FUNCTION_BLOCK Equipo_Motor_No_Rev

VAR_INPUT
PE 	  					  : BOOL; (*Parada deemergencia*)
Lock_Out 				  : BOOL;
Conf_Marcha 			  : BOOL; (*Confirmacion de Marcha *)
Modo_Automatico           : BOOL;
Cmd_Auto         		  : BOOL;
Habilitado  			  : BOOL;
T_Discrepancia            : TIME;
END_VAR

VAR_OUTPUT
	Marcha_Equipo	 	  : BOOL;
	Marcha_Ok  				  : BOOL;
	Estado					  : INT;
	Alr_Discrepancia		  : BOOL;	
	Alr_LockOut        		  : BOOL;
END_VAR

VAR_IN_OUT
	Cmd_Man 				  : BOOL;
	Alarma				      : BOOL;
	Horas_Parciales			  : DINT;
	Horas_Totales		 	  : DINT;
	Reset_Horas         	  : BOOL;
	Reset_Alarma		      : BOOL;
END_VAR

VAR_TEMP
	Reset_Cmd_Auto 		      : BOOL;
	Aux_Limpieza		      : TIME;
END_VAR

VAR_STAT
	Cmd_Auto_Directa		  : BOOL;
	FP_Reset				  : R_TRIG;
	FN_Parada_Auto			  : F_TRIG;
	Parcial_Horas			  : INT;
END_VAR

VAR
	Timer_Discrepancia		  : TON;
	Timer_Segundos		      : TON;
END_VAR
VAR PERSISTENT
	Acionamentos	:UDINT;	//Quantidade de vezes que o motor foi acionado
	TempoFuncionando:UDINT;	//Tempo de funcionamento do motor
		
END_VAR
VAR // added by the converter: edge detectors and wires of the graphical bodies
    _w1, _w2, _w3, _w4, _w5, _w6, _w7, _w8, _w9, _w10 : BOOL;
    _rt1 : R_TRIG;
END_VAR

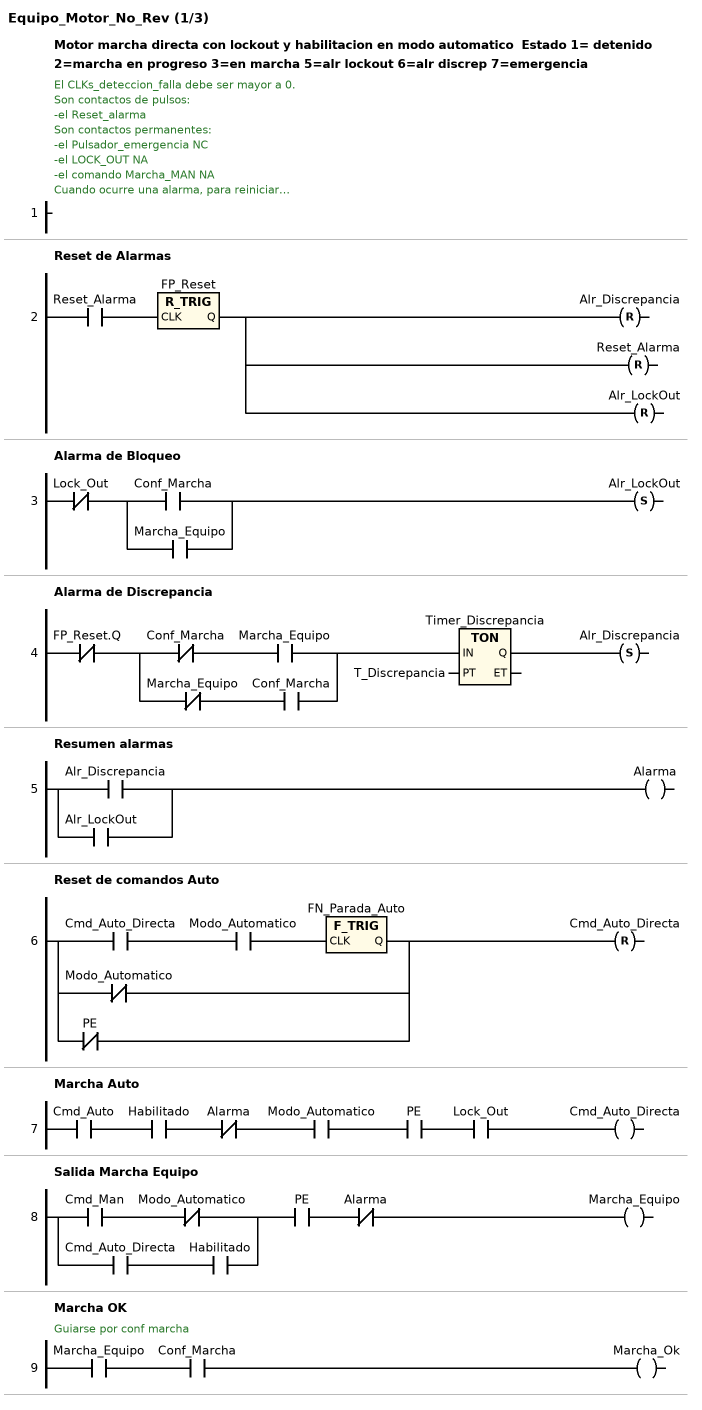
// NETWORK 1: Motor marcha directa con lockout y habilitacion en modo automatico Estado 1= detenido 2=marcha en progreso 3=en marcha 5=alr lockout 6=alr discrep 7=emergencia
// El CLKs_deteccion_falla debe ser mayor a 0.
//
// Son contactos de pulsos:
// -el Reset_alarma
//
// Son contactos permanentes:
// -el Pulsador_emergencia NC
// -el LOCK_OUT NA
// -el comando Marcha_MAN NA
//
// Cuando ocurre una alarma, para reiniciar:
// -en manual reponer la causa de la alarma, pulsar Reset_alarma y pulsar
// Marcha_MAN.
// -en automático reponer la causa de la alarma, pulsar Reset_alarma y si el
// equipo aguas abajo y la Marcha_auto continuan activas, el equipo arrancará.
//
// Siempre que se conmute de automático a manual y viceversa, el equipo se
// detendrá.
//
// Si el equipo es el primero aguas abajo se debe setear siempre en
// 1 Equipos_aguas_abajoOk.
//
// Si el equipo no tiene equipos aguas arribas se debe poner el mismo comando de
// Marcha_MAN en Marcha_aguas_arribaOk

// NETWORK 2: Reset de Alarmas
FP_Reset(CLK := Reset_Alarma); // R_TRIG
Alr_Discrepancia R= FP_Reset.Q;
Reset_Alarma R= FP_Reset.Q;
Alr_LockOut R= FP_Reset.Q;

// NETWORK 3: Alarma de Bloqueo
Alr_LockOut S= NOT Lock_Out AND (Conf_Marcha OR Marcha_Equipo);

// NETWORK 4: Alarma de Discrepancia
Timer_Discrepancia(IN := NOT FP_Reset.Q AND (NOT Conf_Marcha AND Marcha_Equipo OR NOT Marcha_Equipo AND Conf_Marcha), PT := T_Discrepancia); // TON
Alr_Discrepancia S= Timer_Discrepancia.Q;

// NETWORK 5: Resumen alarmas
Alarma := Alr_Discrepancia OR Alr_LockOut;

// NETWORK 6: Reset de comandos Auto
FN_Parada_Auto(CLK := Cmd_Auto_Directa AND Modo_Automatico); // F_TRIG
Cmd_Auto_Directa R= FN_Parada_Auto.Q OR NOT Modo_Automatico OR NOT PE;

// NETWORK 7: Marcha Auto
Cmd_Auto_Directa := Cmd_Auto AND Habilitado AND NOT Alarma AND Modo_Automatico AND PE AND Lock_Out;

// NETWORK 8: Salida Marcha Equipo
Marcha_Equipo := (Cmd_Man AND NOT Modo_Automatico OR Cmd_Auto_Directa AND Habilitado) AND PE AND NOT Alarma;

// NETWORK 9: Marcha OK
// Guiarse por conf marcha
Marcha_Ok := Marcha_Equipo AND Conf_Marcha;

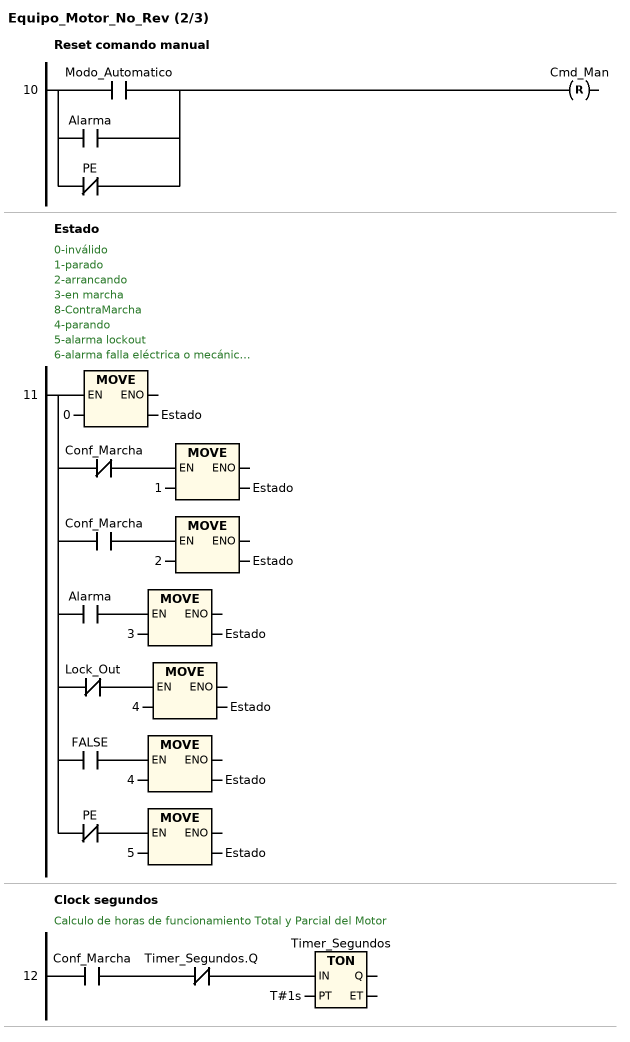
// NETWORK 10: Reset comando manual
Cmd_Man R= Modo_Automatico OR Alarma OR NOT PE;

// NETWORK 11: Estado
// 0-inválido
// 1-parado
// 2-arrancando
// 3-en marcha
// 8-ContraMarcha
// 4-parando
// 5-alarma lockout
// 6-alarma falla eléctrica o mecánica
// 7-alarma pulsador emergencia
Estado := 0;
_w1 := NOT Conf_Marcha;
IF _w1 THEN Estado := 1; END_IF
_w2 := Conf_Marcha;
IF _w2 THEN Estado := 2; END_IF
_w3 := Alarma;
IF _w3 THEN Estado := 3; END_IF
_w4 := NOT Lock_Out;
IF _w4 THEN Estado := 4; END_IF
IF FALSE THEN Estado := 4; END_IF
_w5 := NOT PE;
IF _w5 THEN Estado := 5; END_IF

// NETWORK 12: Clock segundos
// Calculo de horas de funcionamiento Total y Parcial del Motor
Timer_Segundos(IN := Conf_Marcha AND NOT Timer_Segundos.Q, PT := T#1s); // TON

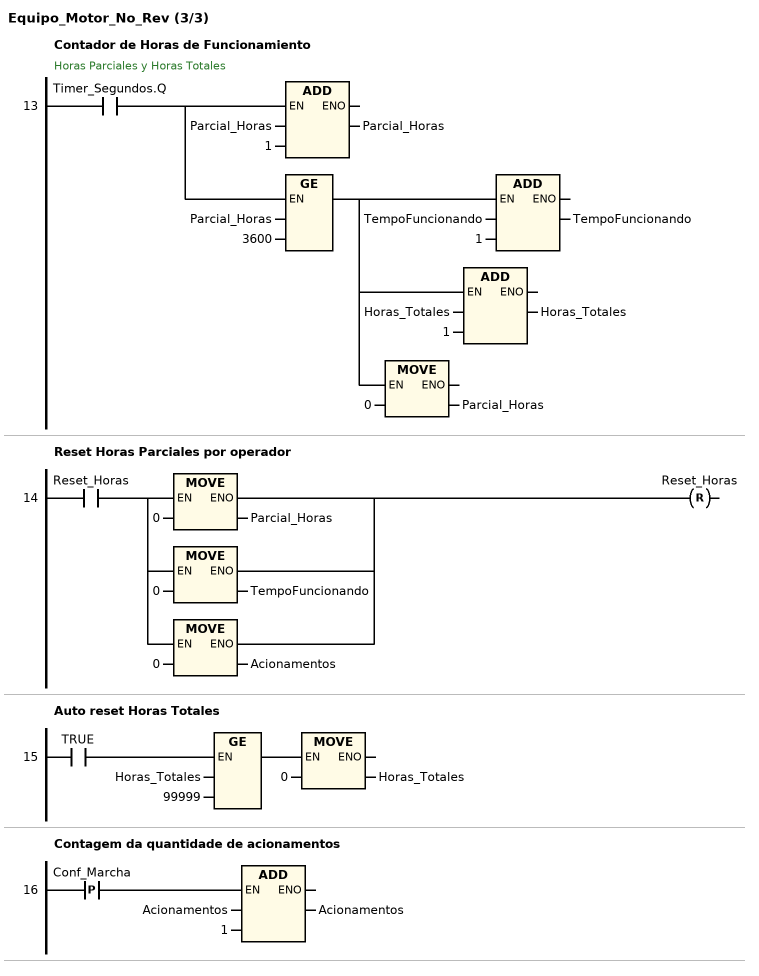
// NETWORK 13: Contador de Horas de Funcionamiento
// Horas Parciales y Horas Totales
_w6 := Timer_Segundos.Q;
IF _w6 THEN Parcial_Horas := Parcial_Horas + 1; END_IF
_w7 := Timer_Segundos.Q AND Parcial_Horas >= 3600;
IF _w7 THEN TempoFuncionando := TempoFuncionando + 1; END_IF
IF _w7 THEN Horas_Totales := Horas_Totales + 1; END_IF
IF _w7 THEN Parcial_Horas := 0; END_IF

// NETWORK 14: Reset Horas Parciales por operador
_w8 := Reset_Horas;
IF _w8 THEN Parcial_Horas := 0; END_IF
_w9 := Reset_Horas;
IF _w9 THEN TempoFuncionando := 0; END_IF
_w10 := Reset_Horas;
IF _w10 THEN Acionamentos := 0; END_IF
Reset_Horas R= _w8 OR (_w9 OR _w10);

// NETWORK 15: Auto reset Horas Totales
IF Horas_Totales >= 99999 THEN Horas_Totales := 0; END_IF

// NETWORK 16: Contagem da quantidade de acionamentos
_rt1(CLK := Conf_Marcha);
IF _rt1.Q THEN Acionamentos := Acionamentos + 1; END_IF

END_FUNCTION_BLOCK

(* stored: Version 1.1.0.1, ProductVersion 3.1.4024.14
   POU Equipo_Motor_No_Rev: Id {98ee8e4a-1dc9-40d8-9da2-89abbee7054b}, SpecialFunc None *)
